FUNCTION_BLOCK FT_GET_GAINS
VAR_INPUT
	TEMP 	: REAL;
	MODE	: BOOL;		// COOLING =0 ; HEATING = 1
END_VAR
VAR_OUTPUT
	//Jacket
	K_P_J 	: REAL;
	K_I_J	: REAL; 
	// Cell
	K_P_C 	: REAL ;		
	K_I_C 	: REAL ;
	K_D_C 	: REAL ;
	//Tracking time 
	T_R_C	: REAL ; 			
	T_R_J	: REAL ; 			
END_VAR
VAR
	TempCase : INT;
END_VAR

IF MODE= TRUE THEN			//HEATING
	IF TEMP < 40 THEN
		TempCase := 3 ;		// 37°C 
	ELSIF TEMP <71 THEN
		TempCase := 3 ;		// up to 71°C 
	ELSIF TEMP <81 THEN
		TempCase := 3 ;		// up to 81°C 
	ELSIF TEMP <91 THEN				
		TempCase := 3 ;		// up to 91°C 
	ELSIF TEMP >115 THEN
		TempCase := 5 ;		// for 121°C
	ELSE
		TempCase := 4 ;		// if over 90°C and below 115 it will handle like 90°C 
	END_IF
ELSE
		TempCase := 0;
END_IF 

CASE TempCase  OF
0:	//COOLING --- till 40°C
	K_P_J := 0.05;
	K_I_J := 1;
	T_R_J := 1;
	
	K_P_C := 7;
	K_I_C := 0.0021;
	//K_D_C := 1050;	
	T_R_C := 21;	
1:  // HEATING ---for 37°C 
	K_P_J := 10;
	K_I_J := 1;
	T_R_J := 1;
	
	K_P_C := 182.5;
	K_I_C := 0.162;
	K_D_C := 385.9;	
	T_R_C := 48.77;	
2:	// HEATING ---for 71°C 
	K_P_J := 0.05;
	K_I_J := 1;
	T_R_J := 1;
	
	K_P_C := 182.5;
	K_I_C := 0.162;
	K_D_C := 385.9;	
	T_R_C := 48.77;
3:	// HEATING ---for 81°C 
	K_P_J := 0.05;
	K_I_J := 1;
	T_R_J := 1;
	
	K_P_C := 62.5;
	K_I_C := 0.06;
	K_D_C := 0;	
	T_R_C := 31.6;	
4:	// HEATING --- for 91°C  ----tbd
	K_P_J := 1;
	K_I_J := 1;
	T_R_J := 1;
	
	K_P_C := 62.5;
	K_I_C := 0.06;
	K_D_C := 0;	
	T_R_C := 31.6;
5:	// STERIL --- for 121°C 

	K_P_C := 0.13;
	K_I_C := 0.0000349;
	K_D_C := 9.28;	
	T_R_C := 515.5;	
END_CASE

END_FUNCTION_BLOCK

(* stored: Version 1.1.0.1, ProductVersion 3.1.4022.12
   POU FT_GET_GAINS: Id {97d12702-10aa-446e-874f-85a6284c0a79}, SpecialFunc None *)
